(* PLC project Untitled1, Beckhoff Automation GmbH TwinCAT PLC Control 3.5.13.21 *)
(* stored: creationDateTime 2024-03-25T12:48:23.9690532, modificationDateTime 2024-03-25T12:48:23.9711951 *)

FUNCTION_BLOCK fbPhoenixTrio
  VAR_INPUT
    IO_In : ARRAY[0..17] OF USINT;
    setChTripPoint : ARRAY[1..8] OF DINT;  (* 0=1A,1=2A,3=3.8A,3=4A,4=6A,5=8A,6=10A *)
    setOnAndReset : ARRAY[1..8] OF BOOL;  (* 0=Off, 1=On/Reset *)
    setChannelPriorityTrip : BOOL;  (* Lowest channel number trips first instead of highest current *)
  END_VAR
  VAR_OUTPUT
    IO_Out : ARRAY[0..6] OF USINT;
    isCurOver90 : BOOL;
    isOutVolt : ARRAY[0..8] OF REAL;  (* 0 is power supply voltage *)
    isOutCur : ARRAY[0..8] OF REAL;  (* 0 is sum of currents *)
    isOutOK : ARRAY[0..8] OF BOOL;
    isOutTripped : ARRAY[1..8] OF BOOL;
  END_VAR

            //Power Supply Status
isCurOver90				:= IO_In[0].3; //Supply over 90% capacity
isOutOK[0]				:= IO_In[0].4=FALSE; //Output not OK inverted
isOutVolt[0]			:= IO_In[1]/10.0; //System Voltage
isOutCur[0]				:= IO_In[3]/10.0; //System Current

//Channel OK Status
isOutOK[1]				:= IO_In[4].6 AND IO_In[4].7=FALSE;
isOutOK[2]				:= IO_In[4].4 AND IO_In[4].5=FALSE;
isOutOK[3]				:= IO_In[4].2 AND IO_In[4].3=FALSE;
isOutOK[4]				:= IO_In[4].0 AND IO_In[4].1=FALSE;
isOutOK[5]				:= IO_In[5].6 AND IO_In[5].7=FALSE;
isOutOK[6]				:= IO_In[5].4 AND IO_In[5].5=FALSE;
isOutOK[7]				:= IO_In[5].2 AND IO_In[5].3=FALSE;
isOutOK[8]				:= IO_In[5].0 AND IO_In[5].1=FALSE;

//Channel Tripped Status
isOutTripped[1]			:= IO_In[4].6 AND IO_In[4].7;
isOutTripped[2]			:= IO_In[4].4 AND IO_In[4].5;
isOutTripped[3]			:= IO_In[4].2 AND IO_In[4].3;
isOutTripped[4]			:= IO_In[4].0 AND IO_In[4].1;
isOutTripped[5]			:= IO_In[5].6 AND IO_In[5].7;
isOutTripped[6]			:= IO_In[5].4 AND IO_In[5].5;
isOutTripped[7]			:= IO_In[5].2 AND IO_In[5].3;
isOutTripped[8]			:= IO_In[5].0 AND IO_In[5].1;

//Voltage and Load
isOutCur[1]				:= IO_In[10]/10.0;//Channel Currents
isOutCur[2]				:= IO_In[11]/10.0;
isOutCur[3]				:= IO_In[12]/10.0;
isOutCur[4]				:= IO_In[13]/10.0;
isOutCur[5]				:= IO_In[14]/10.0;
isOutCur[6]				:= IO_In[15]/10.0;
isOutCur[7]				:= IO_In[16]/10.0;
isOutCur[8]				:= IO_In[17]/10.0;

//Must be true to allow writing of PDO data to PS
IO_Out[0].7				:= 1;

//Trip Point Settings Binary of 0=1A,1=2A,3=3.8A,3=4A,4=6A,5=8A,6=10A
//CH 1
IO_Out[1].3				:= setChTripPoint[1].0;
IO_Out[1].4				:= setChTripPoint[1].1;
IO_Out[1].5				:= setChTripPoint[1].2;
//Ch2
IO_Out[1].0				:= setChTripPoint[2].0;
IO_Out[1].1				:= setChTripPoint[2].1;
IO_Out[1].2				:= setChTripPoint[2].2;
//Ch3
IO_Out[2].3				:= setChTripPoint[3].0;
IO_Out[2].4				:= setChTripPoint[3].1;
IO_Out[2].5				:= setChTripPoint[3].2;
//Ch4
IO_Out[2].0				:= setChTripPoint[4].0;
IO_Out[2].1				:= setChTripPoint[4].1;
IO_Out[2].2				:= setChTripPoint[4].2;
//Ch5
IO_Out[3].3				:= setChTripPoint[5].0;
IO_Out[3].4				:= setChTripPoint[5].1;
IO_Out[3].5				:= setChTripPoint[5].2;
//Ch6
IO_Out[3].0				:= setChTripPoint[6].0;
IO_Out[3].1				:= setChTripPoint[6].1;
IO_Out[3].2				:= setChTripPoint[6].2;
//Ch7
IO_Out[4].3				:= setChTripPoint[7].0;
IO_Out[4].4				:= setChTripPoint[7].1;
IO_Out[4].5				:= setChTripPoint[7].2;
//Ch8
IO_Out[4].0				:= setChTripPoint[8].0;
IO_Out[4].1				:= setChTripPoint[8].1;
IO_Out[4].2				:= setChTripPoint[8].2;

//Sets Current Trip Priority
IO_Out[5].0				:= setChannelPriorityTrip;

//Turns on channel and resets when tripped
IO_Out[6].7				:= setOnAndReset[1] AND isOutTripped[1]=FALSE;
IO_Out[6].6				:= setOnAndReset[2] AND isOutTripped[2]=FALSE;
IO_Out[6].5				:= setOnAndReset[3] AND isOutTripped[3]=FALSE;
IO_Out[6].4				:= setOnAndReset[4] AND isOutTripped[4]=FALSE;
IO_Out[6].3				:= setOnAndReset[5] AND isOutTripped[5]=FALSE;
IO_Out[6].2				:= setOnAndReset[6] AND isOutTripped[6]=FALSE;
IO_Out[6].1				:= setOnAndReset[7] AND isOutTripped[7]=FALSE;
IO_Out[6].0				:= setOnAndReset[8] AND isOutTripped[8]=FALSE;
          
END_FUNCTION_BLOCK
